{attribute 'pack_mode' := '1'}
TYPE ST_MqttAdsShell :
STRUCT
	bNewMessage : BOOL;
	sTopic : STRING(8);
	stMqttPayload : ST_MqttPayload;
END_STRUCT
END_TYPE

(* stored: Version 1.1.0.1, ProductVersion 3.1.4024.0
   DUT ST_MqttAdsShell: Id {0eeb0936-e2e0-4840-992d-149df7d83e34} *)
